(* Logix 5000 project; controller OCV_Tester_EnSG vendor 1 type 14 code 106 rev 32.11; software revision 32.02; part 2 of 2 *)
(* tags used below, declared in another part *)
   AngleLimit : DINT[21];
   AVE_Control : CONTROL;   // battery average ctrl
   battV_avg : DINT;   // battery voltage average
   clearFFO : BOOL;
   contact_t : TIMER[20];
   en_blower : BOOL;
   Failed : BOOL;
   FFOCtrl : CONTROL;
   fifo : DINT;
   hmi_setAngle0 : BOOL;   // set Offset Angle 0
   hmi_setSpeedRef100 : INT;   // hmi_setSpeedRef*100
   index : BOOL;
   lastVolt : DINT;
   MaxV : INT[20];
   OK : BOOL;
   ons : INT;
   pb_SafetyRst : BOOL;   // pb safety reset
   Safety : BOOL;
   StartAngle : DINT;
   tof1s : TIMER;
   ton1s : TIMER;
   unloadBattV : DINT;   // unloaded battV element array
   Angle : DINT;
   battMon : DINT[20];
   battV : DINT[64];
   battV_NOK : INT[21];
   blink1s : BOOL;
   blower0 : BOOL;
   cal_curVoltRaw : INT;
   cal_nom : INT;
   cutOff_thrs : INT;
   DataV : INT[20];
   eStop : BOOL;
   Fault : BOOL;
   FFOMonCtrl : CONTROL;
   FFONOKCtrl : CONTROL;
   FFOPrbNOKCtrl : CONTROL;
   FloatMode : BOOL;
   hmi_accept_thrs : INT;
   hmi_blower0 : BOOL;
   hmi_calMax : BOOL[32];
   hmi_calMin : BOOL[32];
   hmi_contactDur : DINT[20];   // Contact Duration
   hmi_delta : INT;   // float test delta mV
   hmi_setSpeedRef : INT;   // HMI_SetSpeed
   hmi_startingVolt : DINT;   // Init Buffer val
   i : INT;
   idx : DINT;
   NOK : BOOL;
   ons1 : DINT;
   Paused : BOOL;
   probeId_NOK : INT[21];
   probeIdx : INT;   // probe index
   ps_exist : BOOL;
   ps_index : BOOL;
   Reset : BOOL;
   Run : BOOL;
   unloadBattV_NOK : DINT;
   unloadedBattMon : DINT;
   unloadProbe_NOK : INT;
   use_calVal : BOOL;
   V_min : INT;   // detect batt V
   v_rampThrs : INT;
   VMax : INT[20];
   VMin : INT[20];
   volt : INT[20];
(* MainProgram, continued *)

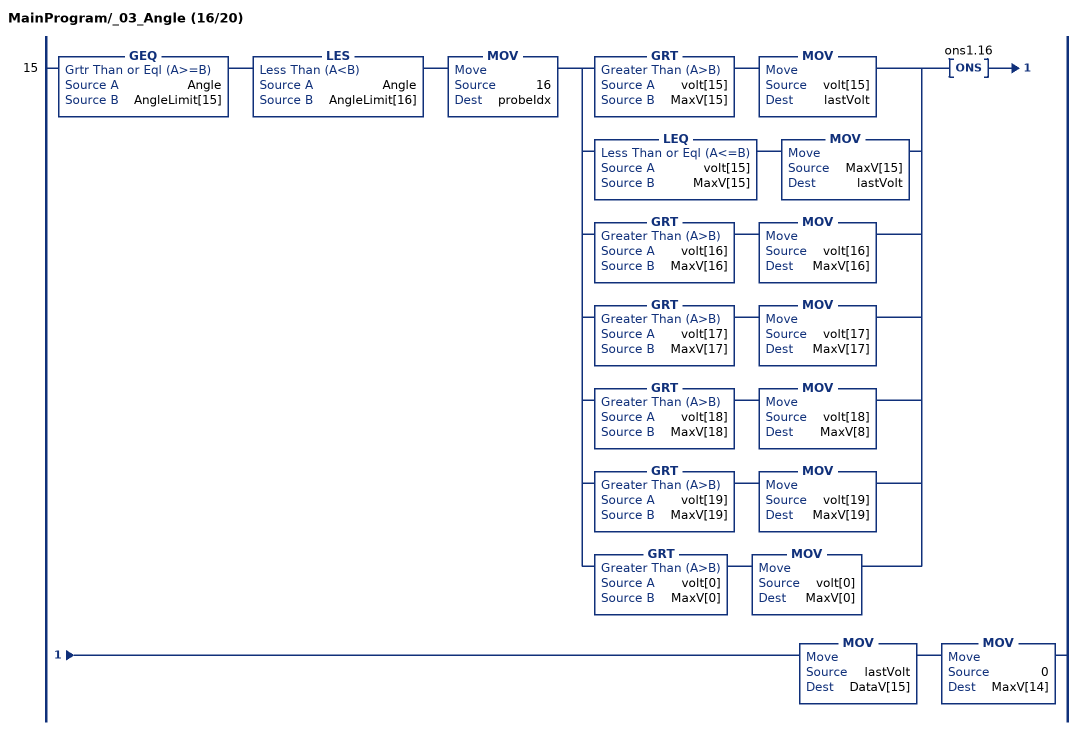
   15: GEQ(Angle,AngleLimit[15])LES(Angle,AngleLimit[16])MOV(16,probeIdx)[GRT(volt[15],MaxV[15]) MOV(volt[15],lastVolt) ,LEQ(volt[15],MaxV[15]) MOV(MaxV[15],lastVolt) ,GRT(volt[16],MaxV[16]) MOV(volt[16],MaxV[16]) ,GRT(volt[17],MaxV[17]) MOV(volt[17],MaxV[17]) ,GRT(volt[18],MaxV[18]) MOV(volt[18],MaxV[8]) ,GRT(volt[19],MaxV[19]) MOV(volt[19],MaxV[19]) ,GRT(volt[0],MaxV[0]) MOV(volt[0],MaxV[0]) ]ONS(ons1.16)MOV(lastVolt,DataV[15])MOV(0,MaxV[14]);
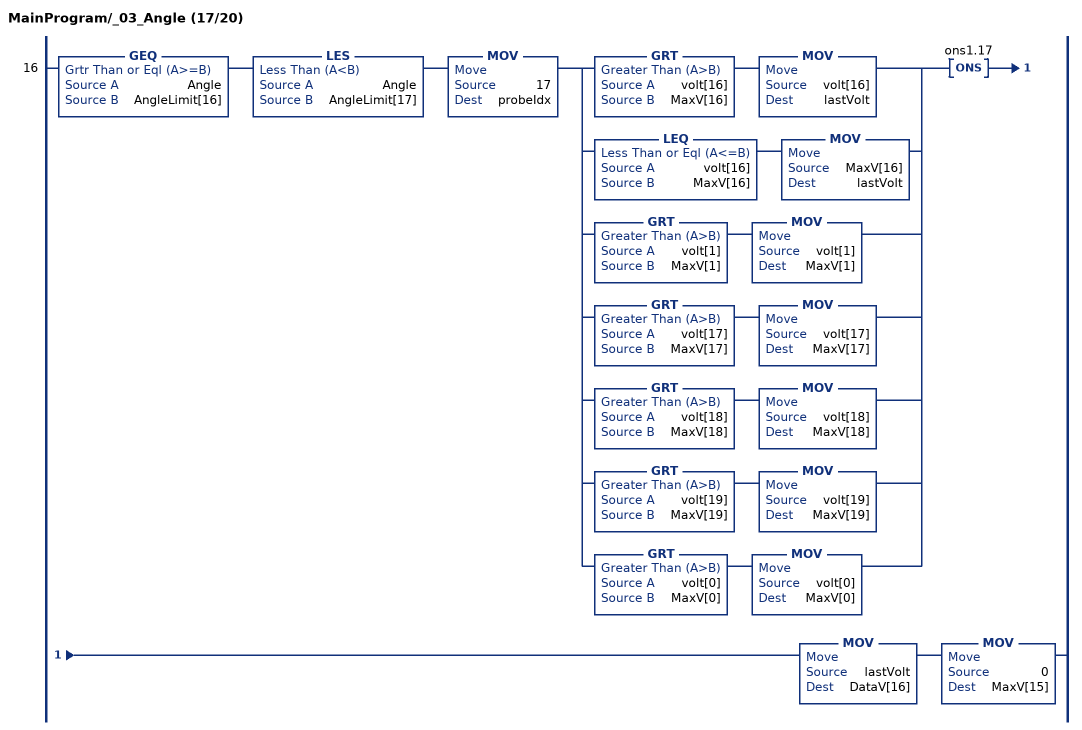
   16: GEQ(Angle,AngleLimit[16])LES(Angle,AngleLimit[17])MOV(17,probeIdx)[GRT(volt[16],MaxV[16]) MOV(volt[16],lastVolt) ,LEQ(volt[16],MaxV[16]) MOV(MaxV[16],lastVolt) ,GRT(volt[1],MaxV[1]) MOV(volt[1],MaxV[1]) ,GRT(volt[17],MaxV[17]) MOV(volt[17],MaxV[17]) ,GRT(volt[18],MaxV[18]) MOV(volt[18],MaxV[18]) ,GRT(volt[19],MaxV[19]) MOV(volt[19],MaxV[19]) ,GRT(volt[0],MaxV[0]) MOV(volt[0],MaxV[0]) ]ONS(ons1.17)MOV(lastVolt,DataV[16])MOV(0,MaxV[15]);
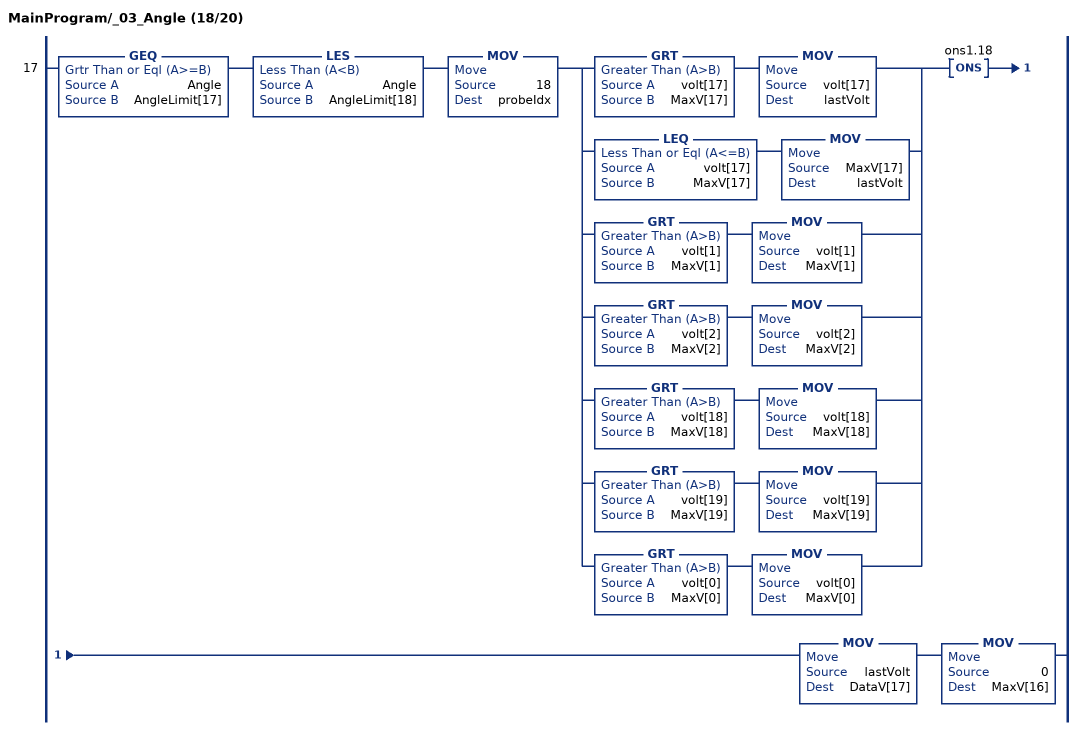
   17: GEQ(Angle,AngleLimit[17])LES(Angle,AngleLimit[18])MOV(18,probeIdx)[GRT(volt[17],MaxV[17]) MOV(volt[17],lastVolt) ,LEQ(volt[17],MaxV[17]) MOV(MaxV[17],lastVolt) ,GRT(volt[1],MaxV[1]) MOV(volt[1],MaxV[1]) ,GRT(volt[2],MaxV[2]) MOV(volt[2],MaxV[2]) ,GRT(volt[18],MaxV[18]) MOV(volt[18],MaxV[18]) ,GRT(volt[19],MaxV[19]) MOV(volt[19],MaxV[19]) ,GRT(volt[0],MaxV[0]) MOV(volt[0],MaxV[0]) ]ONS(ons1.18)MOV(lastVolt,DataV[17])MOV(0,MaxV[16]);
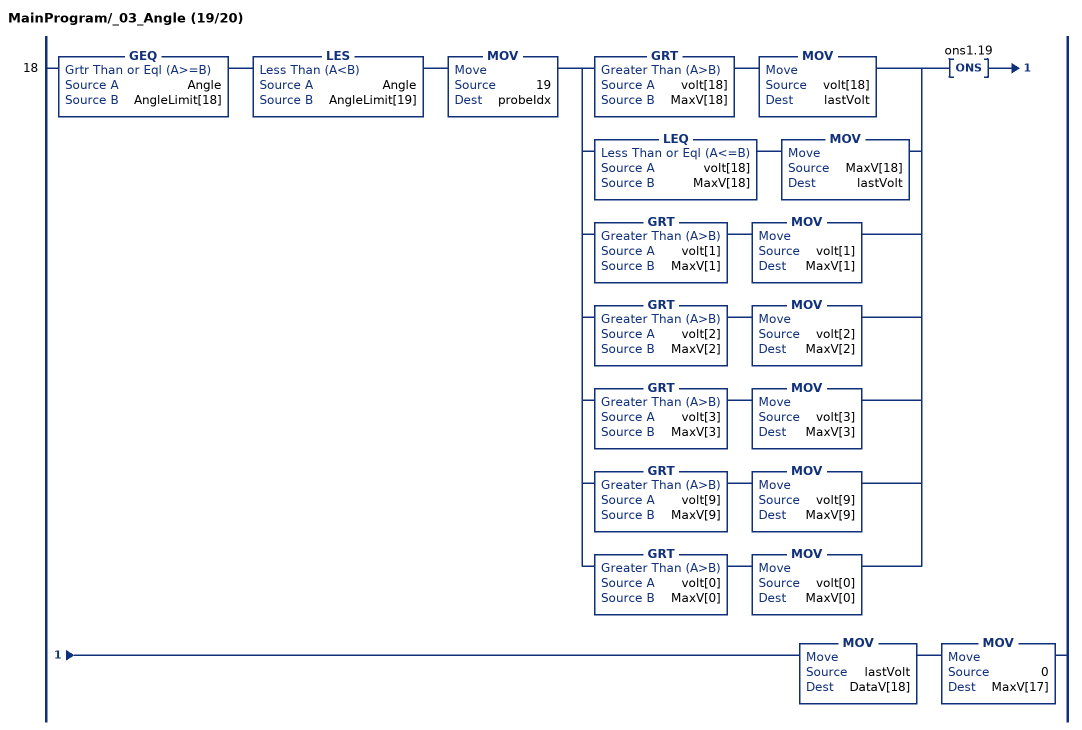
   18: GEQ(Angle,AngleLimit[18])LES(Angle,AngleLimit[19])MOV(19,probeIdx)[GRT(volt[18],MaxV[18]) MOV(volt[18],lastVolt) ,LEQ(volt[18],MaxV[18]) MOV(MaxV[18],lastVolt) ,GRT(volt[1],MaxV[1]) MOV(volt[1],MaxV[1]) ,GRT(volt[2],MaxV[2]) MOV(volt[2],MaxV[2]) ,GRT(volt[3],MaxV[3]) MOV(volt[3],MaxV[3]) ,GRT(volt[9],MaxV[9]) MOV(volt[9],MaxV[9]) ,GRT(volt[0],MaxV[0]) MOV(volt[0],MaxV[0]) ]ONS(ons1.19)MOV(lastVolt,DataV[18])MOV(0,MaxV[17]);
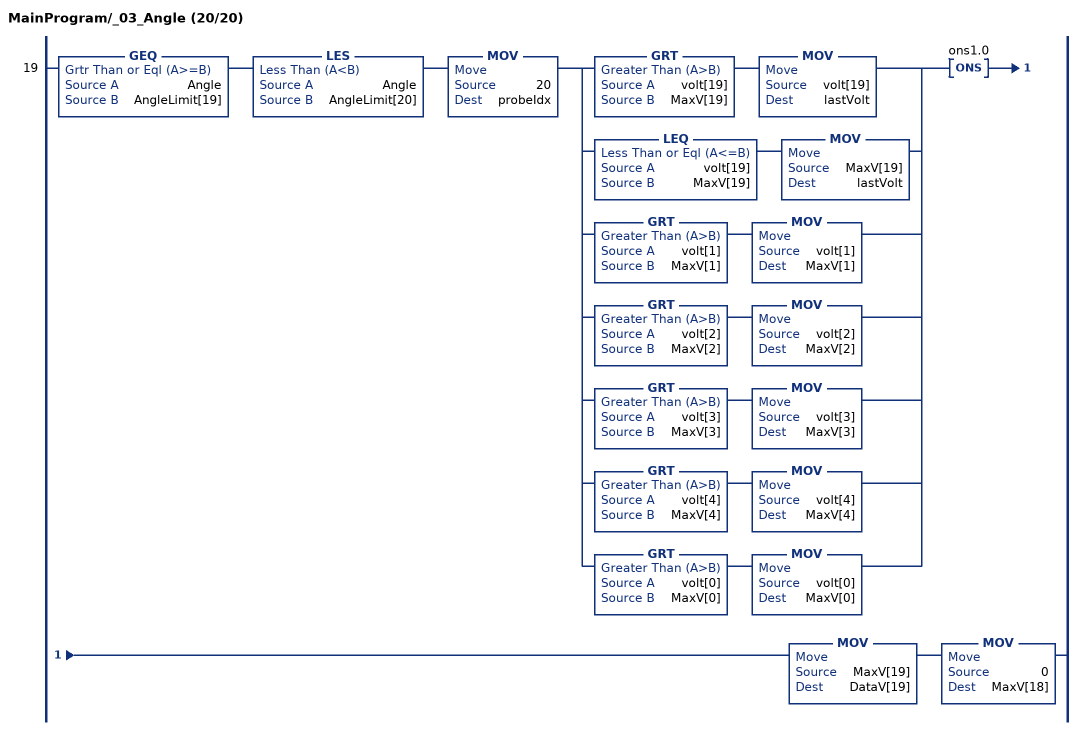
   19: GEQ(Angle,AngleLimit[19])LES(Angle,AngleLimit[20])MOV(20,probeIdx)[GRT(volt[19],MaxV[19]) MOV(volt[19],lastVolt) ,LEQ(volt[19],MaxV[19]) MOV(MaxV[19],lastVolt) ,GRT(volt[1],MaxV[1]) MOV(volt[1],MaxV[1]) ,GRT(volt[2],MaxV[2]) MOV(volt[2],MaxV[2]) ,GRT(volt[3],MaxV[3]) MOV(volt[3],MaxV[3]) ,GRT(volt[4],MaxV[4]) MOV(volt[4],MaxV[4]) ,GRT(volt[0],MaxV[0]) MOV(volt[0],MaxV[0]) ]ONS(ons1.0)MOV(MaxV[19],DataV[19])MOV(0,MaxV[18]);
END_ROUTINE

ROUTINE _04_TestThreshold   (* ladder *)
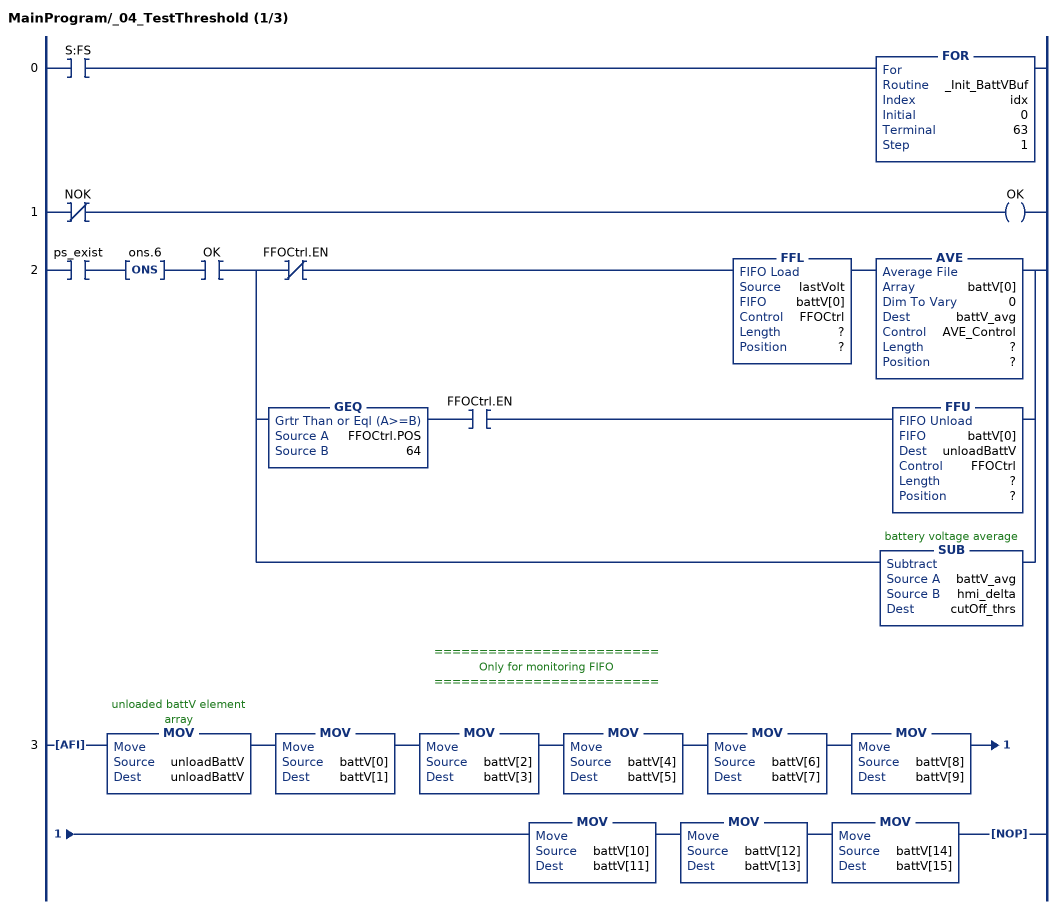
   0: XIC(S:FS)FOR(_Init_BattVBuf,idx,0,63,1);
   1: XIO(NOK)OTE(OK);
   2: XIC(ps_exist)ONS(ons.6)XIC(OK)[XIO(FFOCtrl.EN) FFL(lastVolt,battV[0],FFOCtrl,?,?) AVE(battV[0],0,battV_avg,AVE_Control,?,?) ,GEQ(FFOCtrl.POS,64) XIC(FFOCtrl.EN) FFU(battV[0],unloadBattV,FFOCtrl,?,?) ,SUB(battV_avg,hmi_delta,cutOff_thrs) ];
   // =========================
   // Only for monitoring FIFO
   // =========================
   3: AFI()MOV(unloadBattV,unloadBattV)MOV(battV[0],battV[1])MOV(battV[2],battV[3])MOV(battV[4],battV[5])MOV(battV[6],battV[7])MOV(battV[8],battV[9])MOV(battV[10],battV[11])MOV(battV[12],battV[13])MOV(battV[14],battV[15])NOP();
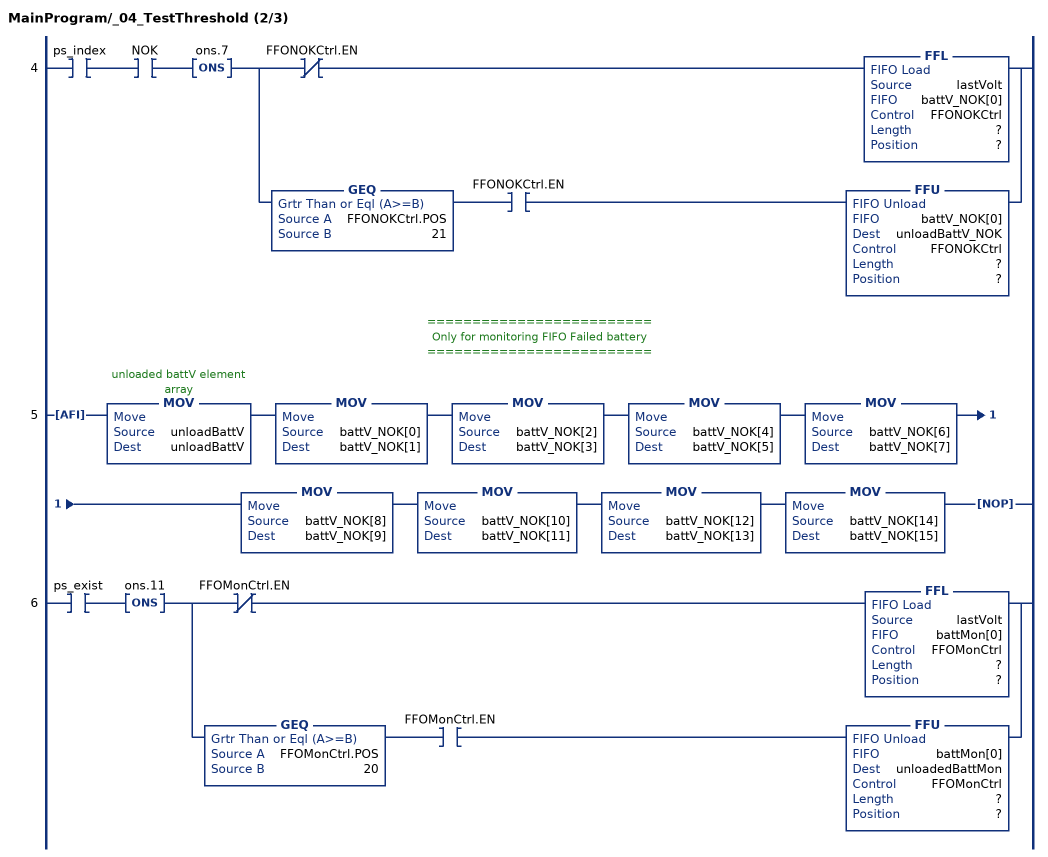
   4: XIC(ps_index)XIC(NOK)ONS(ons.7)[XIO(FFONOKCtrl.EN) FFL(lastVolt,battV_NOK[0],FFONOKCtrl,?,?) ,GEQ(FFONOKCtrl.POS,21) XIC(FFONOKCtrl.EN) FFU(battV_NOK[0],unloadBattV_NOK,FFONOKCtrl,?,?) ];
   // =========================
   // Only for monitoring FIFO Failed battery
   // =========================
   5: AFI()MOV(unloadBattV,unloadBattV)MOV(battV_NOK[0],battV_NOK[1])MOV(battV_NOK[2],battV_NOK[3])MOV(battV_NOK[4],battV_NOK[5])MOV(battV_NOK[6],battV_NOK[7])MOV(battV_NOK[8],battV_NOK[9])MOV(battV_NOK[10],battV_NOK[11])MOV(battV_NOK[12],battV_NOK[13])MOV(battV_NOK[14],battV_NOK[15])NOP();
   6: XIC(ps_exist)ONS(ons.11)[XIO(FFOMonCtrl.EN) FFL(lastVolt,battMon[0],FFOMonCtrl,?,?) ,GEQ(FFOMonCtrl.POS,20) XIC(FFOMonCtrl.EN) FFU(battMon[0],unloadedBattMon,FFOMonCtrl,?,?) ];
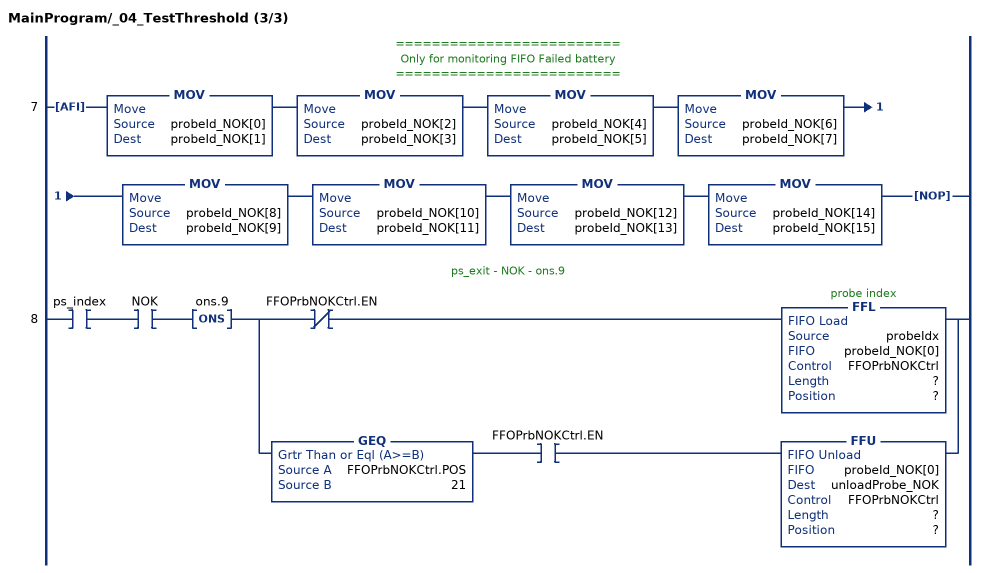
   // =========================
   // Only for monitoring FIFO Failed battery
   // =========================
   7: AFI()MOV(probeId_NOK[0],probeId_NOK[1])MOV(probeId_NOK[2],probeId_NOK[3])MOV(probeId_NOK[4],probeId_NOK[5])MOV(probeId_NOK[6],probeId_NOK[7])MOV(probeId_NOK[8],probeId_NOK[9])MOV(probeId_NOK[10],probeId_NOK[11])MOV(probeId_NOK[12],probeId_NOK[13])MOV(probeId_NOK[14],probeId_NOK[15])NOP();
   // ps_exit - NOK - ons.9
   8: XIC(ps_index)XIC(NOK)ONS(ons.9)[XIO(FFOPrbNOKCtrl.EN) FFL(probeIdx,probeId_NOK[0],FFOPrbNOKCtrl,?,?) ,GEQ(FFOPrbNOKCtrl.POS,21) XIC(FFOPrbNOKCtrl.EN) FFU(probeId_NOK[0],unloadProbe_NOK,FFOPrbNOKCtrl,?,?) ];
END_ROUTINE

ROUTINE _05_Output   (* ladder *)
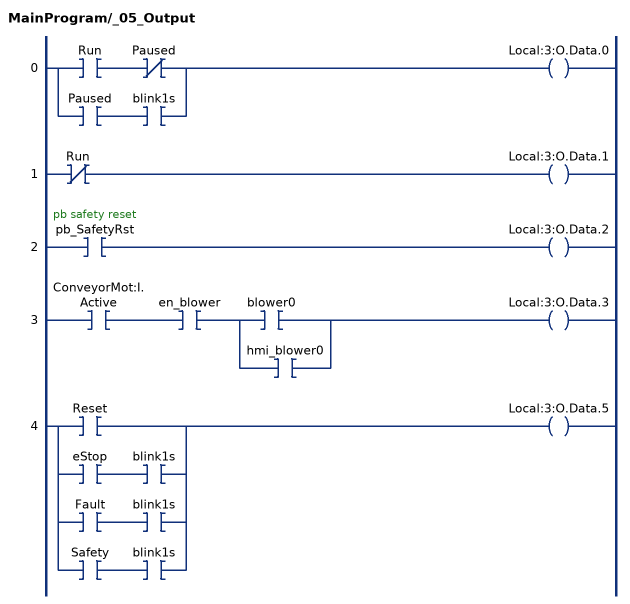
   0: [XIC(Run) XIO(Paused) ,XIC(Paused) XIC(blink1s) ]OTE(Local:3:O.Data.0);
   1: XIO(Run)OTE(Local:3:O.Data.1);
   2: XIC(pb_SafetyRst)OTE(Local:3:O.Data.2);
   3: XIC(ConveyorMot:I.Active)XIC(en_blower)[XIC(blower0) ,XIC(hmi_blower0) ]OTE(Local:3:O.Data.3);
   4: [XIC(Reset) ,XIC(eStop) XIC(blink1s) ,XIC(Fault) XIC(blink1s) ,XIC(Safety) XIC(blink1s) ]OTE(Local:3:O.Data.5);
END_ROUTINE

ROUTINE _07_Settings   (* ladder *)
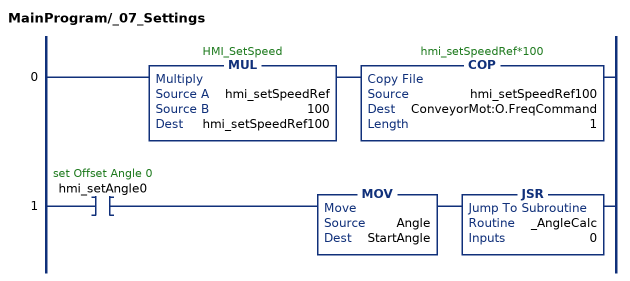
   0: MUL(hmi_setSpeedRef,100,hmi_setSpeedRef100)COP(hmi_setSpeedRef100,ConveyorMot:O.FreqCommand,1);
   1: XIC(hmi_setAngle0)MOV(Angle,StartAngle)JSR(_AngleCalc,0);
END_ROUTINE

ROUTINE _20_Misc   (* ladder *)
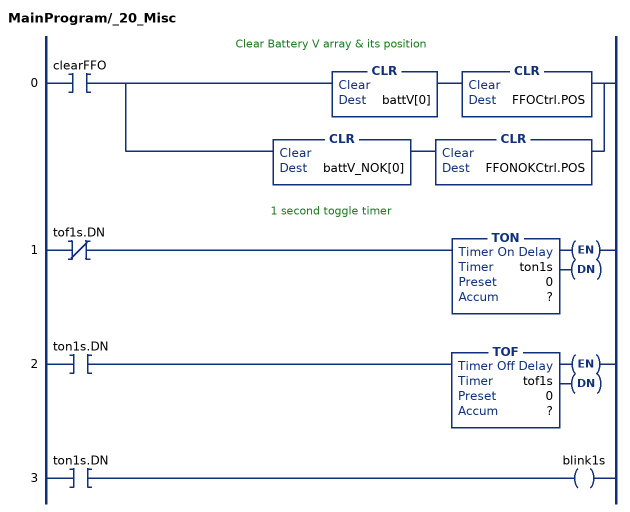
   // Clear Battery V array & its position
   0: XIC(clearFFO)[CLR(battV[0]) CLR(FFOCtrl.POS) ,CLR(battV_NOK[0]) CLR(FFONOKCtrl.POS) ];
   // 1 second toggle timer
   1: XIO(tof1s.DN)TON(ton1s,?,?);
   2: XIC(ton1s.DN)TOF(tof1s,?,?);
   3: XIC(ton1s.DN)OTE(blink1s);
END_ROUTINE

ROUTINE _21_VDuration   (* ladder *)
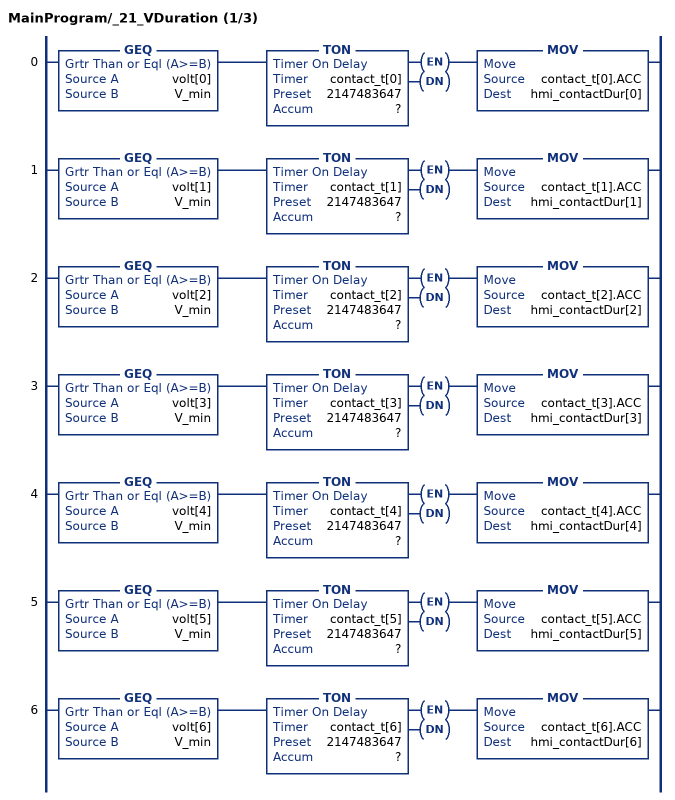
   0: GEQ(volt[0],V_min)TON(contact_t[0],?,?)MOV(contact_t[0].ACC,hmi_contactDur[0]);
   1: GEQ(volt[1],V_min)TON(contact_t[1],?,?)MOV(contact_t[1].ACC,hmi_contactDur[1]);
   2: GEQ(volt[2],V_min)TON(contact_t[2],?,?)MOV(contact_t[2].ACC,hmi_contactDur[2]);
   3: GEQ(volt[3],V_min)TON(contact_t[3],?,?)MOV(contact_t[3].ACC,hmi_contactDur[3]);
   4: GEQ(volt[4],V_min)TON(contact_t[4],?,?)MOV(contact_t[4].ACC,hmi_contactDur[4]);
   5: GEQ(volt[5],V_min)TON(contact_t[5],?,?)MOV(contact_t[5].ACC,hmi_contactDur[5]);
   6: GEQ(volt[6],V_min)TON(contact_t[6],?,?)MOV(contact_t[6].ACC,hmi_contactDur[6]);
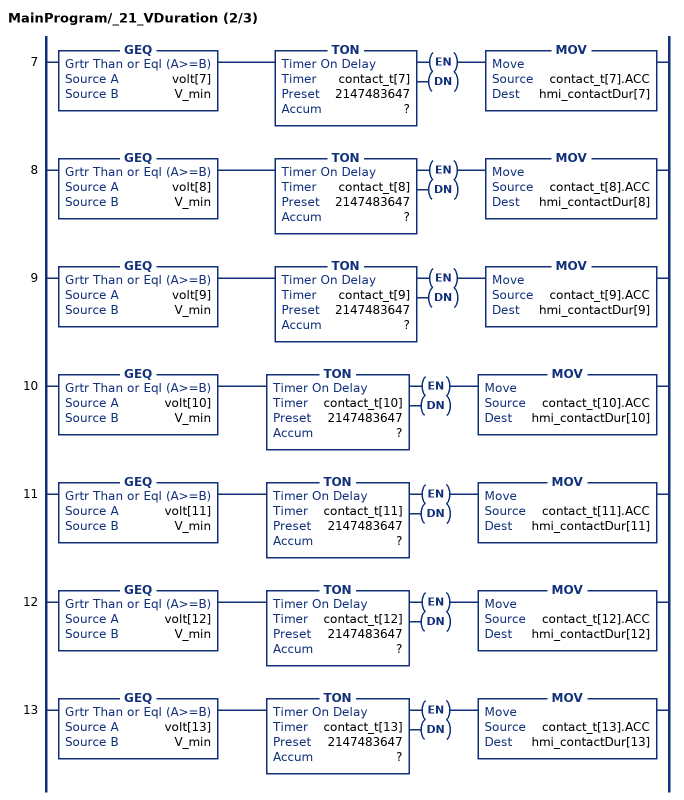
   7: GEQ(volt[7],V_min)TON(contact_t[7],?,?)MOV(contact_t[7].ACC,hmi_contactDur[7]);
   8: GEQ(volt[8],V_min)TON(contact_t[8],?,?)MOV(contact_t[8].ACC,hmi_contactDur[8]);
   9: GEQ(volt[9],V_min)TON(contact_t[9],?,?)MOV(contact_t[9].ACC,hmi_contactDur[9]);
   10: GEQ(volt[10],V_min)TON(contact_t[10],?,?)MOV(contact_t[10].ACC,hmi_contactDur[10]);
   11: GEQ(volt[11],V_min)TON(contact_t[11],?,?)MOV(contact_t[11].ACC,hmi_contactDur[11]);
   12: GEQ(volt[12],V_min)TON(contact_t[12],?,?)MOV(contact_t[12].ACC,hmi_contactDur[12]);
   13: GEQ(volt[13],V_min)TON(contact_t[13],?,?)MOV(contact_t[13].ACC,hmi_contactDur[13]);
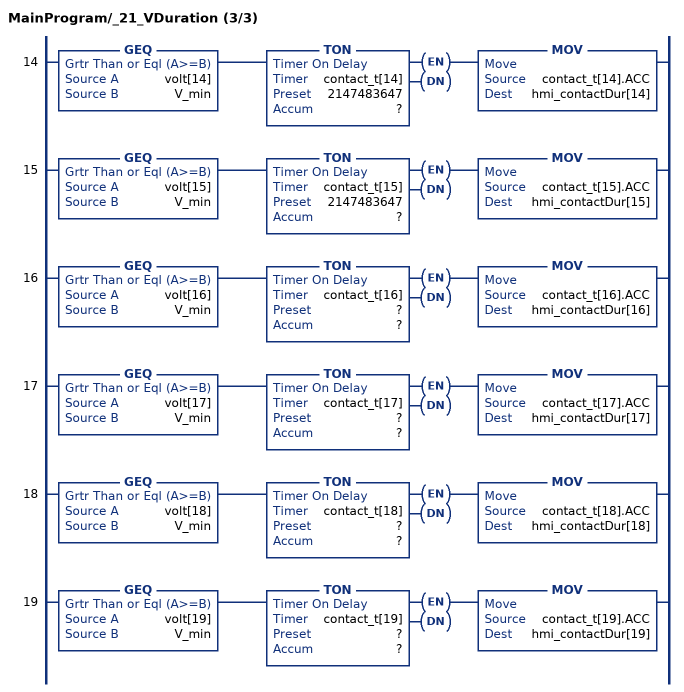
   14: GEQ(volt[14],V_min)TON(contact_t[14],?,?)MOV(contact_t[14].ACC,hmi_contactDur[14]);
   15: GEQ(volt[15],V_min)TON(contact_t[15],?,?)MOV(contact_t[15].ACC,hmi_contactDur[15]);
   16: GEQ(volt[16],V_min)TON(contact_t[16],?,?)MOV(contact_t[16].ACC,hmi_contactDur[16]);
   17: GEQ(volt[17],V_min)TON(contact_t[17],?,?)MOV(contact_t[17].ACC,hmi_contactDur[17]);
   18: GEQ(volt[18],V_min)TON(contact_t[18],?,?)MOV(contact_t[18].ACC,hmi_contactDur[18]);
   19: GEQ(volt[19],V_min)TON(contact_t[19],?,?)MOV(contact_t[19].ACC,hmi_contactDur[19]);
END_ROUTINE

ROUTINE _AngleCalc   (* structured text *)
   AngleLimit[0] := StartAngle;
   AngleLimit[1] := StartAngle + 18*1;
   AngleLimit[2] := StartAngle + 18*2;
   AngleLimit[3] := StartAngle + 18*3;
   AngleLimit[4] := StartAngle + 18*4;
   AngleLimit[5] := StartAngle + 18*5;
   AngleLimit[6] := StartAngle + 18*6;
   AngleLimit[7] := StartAngle + 18*7;
   AngleLimit[8] := StartAngle + 18*8;
   AngleLimit[9] := StartAngle + 18*9;
   AngleLimit[10] := StartAngle + 18*10;
   AngleLimit[11] := StartAngle + 18*11;
   AngleLimit[12] := StartAngle + 18*12;
   AngleLimit[13] := StartAngle + 18*13;
   AngleLimit[14] := StartAngle + 18*14;
   AngleLimit[15] := StartAngle + 18*15;
   AngleLimit[16] := StartAngle + 18*16;
   AngleLimit[17] := StartAngle + 18*17;
   AngleLimit[18] := StartAngle + 18*18;
   AngleLimit[19] := StartAngle + 18*19;
   AngleLimit[20] := StartAngle + 18*20;
   if AngleLimit[1] > 360 then
   	AngleLimit[1] := AngleLimit[1] - 360;
   end_if;
   if AngleLimit[2] > 360 then
   	AngleLimit[2] := AngleLimit[2] - 360;
   end_if;
   if AngleLimit[3] > 360 then
   	AngleLimit[3] := AngleLimit[3] - 360;
   end_if;
   if AngleLimit[4] > 360 then
   	AngleLimit[4] := AngleLimit[4] - 360;
   end_if;
   if AngleLimit[5] > 360 then
   	AngleLimit[5] := AngleLimit[5] - 360;
   end_if;
   if AngleLimit[6] > 360 then
   	AngleLimit[6] := AngleLimit[6] - 360;
   end_if;
   if AngleLimit[7] > 360 then
   	AngleLimit[7] := AngleLimit[7] - 360;
   end_if;
   if AngleLimit[8] > 360 then
   	AngleLimit[8] := AngleLimit[8] - 360;
   end_if;
   if AngleLimit[9] > 360 then
   	AngleLimit[9] := AngleLimit[9] - 360;
   end_if;
   if AngleLimit[10] > 360 then
   	AngleLimit[10] := AngleLimit[10] - 360;
   end_if;
   if AngleLimit[11] > 360 then
   	AngleLimit[11] := AngleLimit[11] - 360;
   end_if;
   if AngleLimit[12] > 360 then
   	AngleLimit[12] := AngleLimit[12] - 360;
   end_if;
   if AngleLimit[13] > 360 then
   	AngleLimit[13] := AngleLimit[13] - 360;
   end_if;
   if AngleLimit[14] > 360 then
   	AngleLimit[14] := AngleLimit[14] - 360;
   end_if;
   if AngleLimit[15] > 360 then
   	AngleLimit[15] := AngleLimit[15] - 360;
   end_if;
   if AngleLimit[16] > 360 then
   	AngleLimit[16] := AngleLimit[16] - 360;
   end_if;
   if AngleLimit[16] > 360 then
   	AngleLimit[16] := AngleLimit[16] - 360;
   end_if;
   if AngleLimit[17] > 360 then
   	AngleLimit[17] := AngleLimit[17] - 360;
   end_if;
   if AngleLimit[18] > 360 then
   	AngleLimit[18] := AngleLimit[18] - 360;
   end_if;
   if AngleLimit[19] > 360 then
   	AngleLimit[19] := AngleLimit[19] - 360;
   end_if;
   if AngleLimit[20] > 360 then
   	AngleLimit[20] := AngleLimit[20] - 360;
   end_if;
END_ROUTINE

ROUTINE _Init_BattVBuf   (* ladder *)
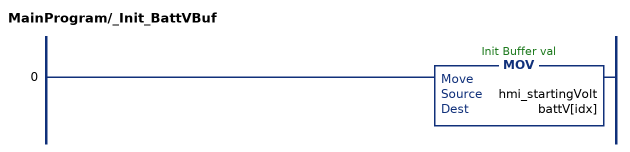
   0: MOV(hmi_startingVolt,battV[idx]);
END_ROUTINE

ROUTINE _onIndex   (* structured text *)
   
   if lastVolt <> 0 then
   
   	if FloatMode then
   		if lastVolt <= cutOff_thrs or lastVolt < hmi_accept_thrs then
   			NOK := 1;
   
   		else
   			NOK := 0;
   		end_if;
   	else
   		if lastVolt <= hmi_accept_thrs then
   			NOK := 1;
   		else
   			NOK := 0;
   		end_if;
   	end_if;
   else
   	NOK:= 0;
   end_if;
END_ROUTINE

ROUTINE AI_Convert   (* structured text *)
   (*
   	This is to plot and manipulate analog input into local variable volt [20]
   	Due to the pull up behaviour of IF16V module
   *)
   
   // cal_nom is real volt difference : 2V - 0V : 2000 mv
   // VMax is the 2V value from AI register
   // VMin is the 0V value from AI register
   // Calibrated Value = (VmaxReal- VminReal)/ (VMax - VMin) * Volt_now
   
   // volt[0] := (cal_nom)/(VMax[0] - VMin[0]) * Local:5:I.Ch00Data;
   
   if Local:5:I.Ch00Data > v_rampThrs then
   	(*if (5250 - Local:5:I.Ch00Data) < v_rampThrs then
   		volt[0] := 5250 - Local:5:I.Ch00Data;
   	end_if;*)
   	volt[0] := 0;
   	volt[10] := 0;
   else
   	if use_calVal then
   		volt[0] := (cal_nom)/(VMax[0] - VMin[0]) * Local:5:I.Ch00Data;
   		volt[10] := (cal_nom)/(VMax[0] - VMin[0]) * Local:5:I.Ch00Data;
   
   	else
   		volt[0] := Local:5:I.Ch00Data;
   		volt[10] := Local:5:I.Ch00Data;
   	end_if;
   end_if;
   if Local:5:I.Ch01Data > v_rampThrs then
   	volt[1] := 0;
   	volt[11] := 0;
   else
   	if use_calVal then
   		volt[1] := (cal_nom)/(VMax[1] - VMin[1]) * Local:5:I.Ch01Data;
   		volt[11] := (cal_nom)/(VMax[1] - VMin[1]) * Local:5:I.Ch01Data;
   	else
   		volt[1] := Local:5:I.Ch01Data;
   		volt[11] := Local:5:I.Ch01Data;
   	end_if;
   end_if;
   if Local:5:I.Ch02Data > v_rampThrs then
   	volt[2] := 0;
   	volt[12] := 0;
   else
   	if use_calVal then
   		volt[2] := (cal_nom)/(VMax[2] - VMin[2]) * Local:5:I.Ch02Data;
   		volt[12] := (cal_nom)/(VMax[2] - VMin[2]) * Local:5:I.Ch02Data;
   	else
   		volt[2] := Local:5:I.Ch02Data;
   		volt[12] := Local:5:I.Ch02Data;
   	end_if;
   end_if;
   if Local:5:I.Ch03Data > v_rampThrs then
   	volt[3] := 0;
   	volt[13] := 0;
   
   else
   	if use_calVal then
   		volt[3] := (cal_nom)/(VMax[3] - VMin[3]) * Local:5:I.Ch03Data;
   		volt[13] := (cal_nom)/(VMax[3] - VMin[3]) * Local:5:I.Ch03Data;
   	else
   		volt[3] := Local:5:I.Ch03Data;
   		volt[13] := Local:5:I.Ch03Data;
   	end_if;
   end_if;
   if Local:5:I.Ch04Data > v_rampThrs then
   	volt[4] := 0;
   	volt[14] := 0;
   else
   	if use_calVal then
   		volt[4] := (cal_nom)/(VMax[4] - VMin[4]) * Local:5:I.Ch04Data;
   		volt[14] := (cal_nom)/(VMax[4] - VMin[4]) * Local:5:I.Ch04Data;
   	else
   		volt[4] := Local:5:I.Ch04Data;
   		volt[14] := Local:5:I.Ch04Data;
   	end_if;
   end_if;
   if Local:5:I.Ch05Data > v_rampThrs then
   	volt[5] := 0;
   	volt[15] := 0;
   else
   	if use_calVal then
   		volt[5] := (cal_nom)/(VMax[5] - VMin[5]) * Local:5:I.Ch05Data;
   		volt[15] := (cal_nom)/(VMax[5] - VMin[5]) * Local:5:I.Ch05Data;
   	else
   		volt[5] := Local:5:I.Ch05Data;
   		volt[15] := Local:5:I.Ch05Data;
   	end_if;
   end_if;
   if Local:5:I.Ch06Data > v_rampThrs then
   	volt[6] := 0;
   	volt[16] := 0;
   else
   	if use_calVal then
   		volt[6] := (cal_nom)/(VMax[6] - VMin[6]) * Local:5:I.Ch06Data;
   		volt[16] := (cal_nom)/(VMax[6] - VMin[6]) * Local:5:I.Ch06Data;
   	else
   		volt[6] := Local:5:I.Ch06Data;
   		volt[16] := Local:5:I.Ch06Data;
   	end_if;
   end_if;
   
   // Due to problem suspection on Local:5:I.Ch07Data, index 7-9 (8-10 real) is put on Local:5:I.Ch8Data to Ch10Data
   
   if Local:5:I.Ch08Data > v_rampThrs then
   	volt[7] := 0;
   	volt[17] := 0;
   else
   	if use_calVal then
   		volt[7] := (cal_nom)/(VMax[8] - VMin[8]) * Local:5:I.Ch08Data;
   		volt[17] := (cal_nom)/(VMax[8] - VMin[8]) * Local:5:I.Ch08Data;
   	else
   		volt[7] := Local:5:I.Ch08Data;
   		volt[17] := Local:5:I.Ch08Data;
   	end_if;
   end_if;
   if Local:5:I.Ch09Data > v_rampThrs then
   	volt[8] := 0;
   	volt[18] := 0;
   else
   	if use_calVal then
   		volt[8] := (cal_nom)/(VMax[9] - VMin[9]) * Local:5:I.Ch09Data;
   		volt[18] := (cal_nom)/(VMax[9] - VMin[9]) * Local:5:I.Ch09Data;
   	else
   		volt[8] := Local:5:I.Ch09Data;
   		volt[18] := Local:5:I.Ch09Data;
   	end_if;
   end_if;
   if Local:5:I.Ch10Data > v_rampThrs then
   	volt[9] := 0;
   	volt[19] := 0;
   else
   	if use_calVal then
   		volt[9] := (cal_nom)/(VMax[10] - VMin[10]) * Local:5:I.Ch10Data;
   		volt[19] := (cal_nom)/(VMax[10] - VMin[10]) * Local:5:I.Ch10Data;
   	else
   		volt[9] := Local:5:I.Ch10Data;
   		volt[19] := Local:5:I.Ch10Data;
   	end_if;
   end_if;
   
   (*
   if Local:5:I.Ch11Data > v_rampThrs then
   	volt[11] := 0;
   else
   	if use_calVal then
   		volt[11] := (cal_nom)/(VMax[11] - VMin[11]) * Local:5:I.Ch11Data;
   	else
   		volt[11] := Local:5:I.Ch11Data;
   	end_if;
   end_if;
   if Local:5:I.Ch12Data > v_rampThrs then
   	volt[12] := 0;
   else
   	if use_calVal then
   		volt[12] := (cal_nom)/(VMax[12] - VMin[12]) * Local:5:I.Ch12Data;
   	else
   		volt[12] := Local:5:I.Ch12Data;
   	end_if;
   end_if;
   if Local:5:I.Ch13Data > v_rampThrs then
   	volt[13] := 0;
   else
   	if use_calVal then
   		volt[13] := (cal_nom)/(VMax[13] - VMin[13]) * Local:5:I.Ch13Data;
   	else
   		volt[13] := Local:5:I.Ch13Data;
   	end_if;
   end_if;
   if Local:5:I.Ch14Data > v_rampThrs then
   	volt[14] := 0;
   else
   	if use_calVal then
   		volt[14] := (cal_nom)/(VMax[14] - VMin[14]) * Local:5:I.Ch14Data;
   	else
   		volt[14] := Local:5:I.Ch14Data;
   	end_if;
   end_if;
   if Local:5:I.Ch15Data > v_rampThrs then
   	volt[15] := 0;
   else
   	if use_calVal then
   		volt[15] := (cal_nom)/(VMax[15] - VMin[15]) * Local:5:I.Ch15Data;
   	else
   		volt[15] := Local:5:I.Ch15Data;
   	end_if;
   end_if;
   
   // Module IF8
   if Local:4:I.Ch0Data < 80 then
   	volt[16] := 0;
   else
   	if use_calVal then
   		volt[16] := (cal_nom)/(VMax[16] - VMin[16]) * Local:4:I.Ch0Data;
   	else
   		volt[16] := Local:4:I.Ch0Data;
   	end_if;
   end_if;
   if Local:4:I.Ch1Data < 80 then
   	volt[17] := 0;
   else
   	if use_calVal then
   		volt[17] := (cal_nom)/(VMax[17] - VMin[17]) * Local:4:I.Ch1Data;
   	else
   		volt[17] := Local:4:I.Ch1Data;
   	end_if;
   end_if;
   if Local:4:I.Ch2Data < 80 then
   	volt[18] := 0;
   else
   	if use_calVal then
   		volt[18] := (cal_nom)/(VMax[18] - VMin[18]) * Local:4:I.Ch2Data;
   	else
   		volt[18] := Local:4:I.Ch2Data;
   	end_if;
   end_if;
   if Local:4:I.Ch3Data < 80 then
   	volt[19] := 0;
   else
   	if use_calVal then
   		volt[19] := (cal_nom)/(VMax[19] - VMin[19]) * Local:4:I.Ch3Data;
   	else
   		volt[19] := Local:4:I.Ch3Data;
   	end_if;
   end_if;
   
   // Due to problem suspection on Local:5:I.Ch07Data, index 7 (8 real) is put on Local:4:I.Ch4Data
   if Local:4:I.Ch4Data < 80 then
   	volt[7] := 0;
   else
   	if use_calVal then
   		volt[7] := (cal_nom)/(VMax[7] - VMin[7]) * Local:4:I.Ch4Data;
   	else
   		volt[7] := Local:4:I.Ch4Data;
   	end_if;
   end_if;
   *)
END_ROUTINE

ROUTINE Calibration   (* structured text *)
   
   if hmi_calMax[0] then
   	VMax[0] := Local:5:I.Ch00Data;
   end_if;
   if hmi_calMin[0] then
   	VMin[0] := Local:5:I.Ch00Data;
   end_if;
   
   if hmi_calMax[1] then
   	VMax[1] := Local:5:I.Ch01Data;
   end_if;
   if hmi_calMin[1] then
   	VMin[1] := Local:5:I.Ch01Data;
   end_if;
   
   if hmi_calMax[2] then
   	VMax[2] := Local:5:I.Ch02Data;
   end_if;
   if hmi_calMin[2] then
   	VMin[2] := Local:5:I.Ch02Data;
   end_if;
   
   if hmi_calMax[3] then
   	VMax[3] := Local:5:I.Ch03Data;
   end_if;
   if hmi_calMin[3] then
   	VMin[3] := Local:5:I.Ch03Data;
   end_if;
   
   if hmi_calMax[4] then
   	VMax[4] := Local:5:I.Ch04Data;
   end_if;
   if hmi_calMin[4] then
   	VMin[4] := Local:5:I.Ch04Data;
   end_if;
   
   if hmi_calMax[5] then
   	VMax[5] := Local:5:I.Ch05Data;
   end_if;
   if hmi_calMin[5] then
   	VMin[5] := Local:5:I.Ch05Data;
   end_if;
   
   if hmi_calMax[6] then
   	VMax[6] := Local:5:I.Ch06Data;
   end_if;
   if hmi_calMin[6] then
   	VMin[6] := Local:5:I.Ch06Data;
   end_if;
   
   if hmi_calMax[7] then
   	VMax[7] := Local:5:I.Ch07Data;
   end_if;
   if hmi_calMin[7] then
   	VMin[7] := Local:5:I.Ch07Data;
   end_if;
   
   if hmi_calMax[8] then
   	VMax[8] := Local:5:I.Ch08Data;
   end_if;
   if hmi_calMin[8] then
   	VMin[8] := Local:5:I.Ch08Data;
   end_if;
   
   if hmi_calMax[9] then
   	VMax[9] := Local:5:I.Ch09Data;
   end_if;
   if hmi_calMin[9] then
   	VMin[9] := Local:5:I.Ch09Data;
   end_if;
   (*
   if hmi_calMax[10] then
   	VMax[10] := Local:5:I.Ch10Data;
   	cal_curVoltRaw := VMax[10];
   end_if;
   if hmi_calMin[10] then
   	VMin[10] := Local:5:I.Ch10Data;
   	cal_curVoltRaw := VMin[10];
   end_if;
   
   if hmi_calMax[11] then
   	VMax[11] := Local:5:I.Ch11Data;
   	cal_curVoltRaw := VMax[11];
   end_if;
   if hmi_calMin[11] then
   	VMin[11] := Local:5:I.Ch11Data;
   	cal_curVoltRaw := VMin[11];
   end_if;
   
   if hmi_calMax[12] then
   	VMax[12] := Local:5:I.Ch12Data;
   	cal_curVoltRaw := VMax[12];
   end_if;
   if hmi_calMin[12] then
   	VMin[12] := Local:5:I.Ch12Data;
   	cal_curVoltRaw := VMin[12];
   end_if;
   
   if hmi_calMax[13] then
   	VMax[13] := Local:5:I.Ch13Data;
   	cal_curVoltRaw := VMax[13];
   end_if;
   if hmi_calMin[13] then
   	VMin[13] := Local:5:I.Ch13Data;
   	cal_curVoltRaw := VMin[13];
   end_if;
   
   if hmi_calMax[14] then
   	VMax[14] := Local:5:I.Ch14Data;
   	cal_curVoltRaw := VMax[14];
   end_if;
   if hmi_calMin[14] then
   	VMin[14] := Local:5:I.Ch14Data;
   	cal_curVoltRaw := VMin[14];
   end_if;
   
   if hmi_calMax[15] then
   	VMax[15] := Local:5:I.Ch15Data;
   	cal_curVoltRaw := VMax[15];
   end_if;
   if hmi_calMin[15] then
   	VMin[15] := Local:5:I.Ch15Data;
   	cal_curVoltRaw := VMin[15];
   end_if;
   
   if hmi_calMax[16] then
   	VMax[16] := Local:4:I.Ch0Data;
   	cal_curVoltRaw := VMax[16];
   end_if;
   if hmi_calMin[16] then
   	VMin[16] := Local:4:I.Ch0Data;
   	cal_curVoltRaw := VMin[16];
   end_if;
   
   if hmi_calMax[17] then
   	VMax[17] := Local:4:I.Ch1Data;
   	cal_curVoltRaw := VMax[17];
   end_if;
   if hmi_calMin[17] then
   	VMin[17] := Local:4:I.Ch1Data;
   	cal_curVoltRaw := VMin[17];
   end_if;
   
   if hmi_calMax[18] then
   	VMax[18] := Local:4:I.Ch2Data;
   	cal_curVoltRaw := VMax[18];
   end_if;
   if hmi_calMin[18] then
   	VMin[18] := Local:4:I.Ch2Data;
   	cal_curVoltRaw := VMin[18];
   end_if;
   
   if hmi_calMax[19] then
   	VMax[19] := Local:4:I.Ch3Data;
   	cal_curVoltRaw := VMax[19];
   end_if;
   if hmi_calMin[19] then
   	VMin[19] := Local:4:I.Ch3Data;
   	cal_curVoltRaw := VMin[19];
   end_if;
   *)
END_ROUTINE

ROUTINE MainRoutine   (* ladder *)
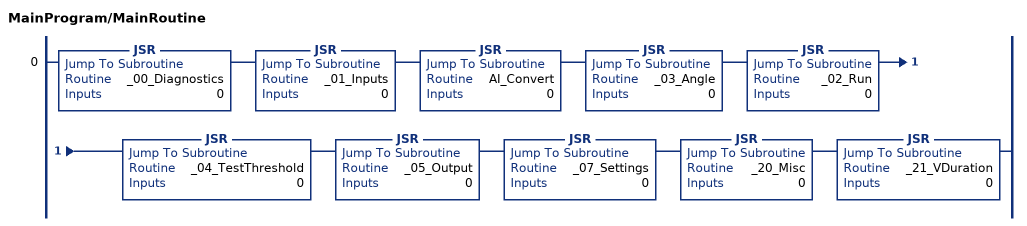
   0: JSR(_00_Diagnostics,0)JSR(_01_Inputs,0)JSR(AI_Convert,0)JSR(_03_Angle,0)JSR(_02_Run,0)JSR(_04_TestThreshold,0)JSR(_05_Output,0)JSR(_07_Settings,0)JSR(_20_Misc,0)JSR(_21_VDuration,0);
END_ROUTINE
END_PROGRAM
